TYPE ST_HW_OutputsInOutFeed :
STRUCT
	OKToRemove			: BOOL; //Indication that pallet is ok to remove
	OKToDeposit			: BOOL; //Indication that pallet is ok to add
	Drive_Run_UpDown	: BOOL; //Drive run lift up/down
END_STRUCT
END_TYPE

(* stored: Version 1.1.0.1, ProductVersion 3.1.4024.9
   DUT ST_HW_OutputsInOutFeed: Id {8955c274-d231-4bf2-b052-c59f4a9c11fe} *)
